// TIA Portal project "5 Run - 2 Stop (2T)" (V16)

(* hardware
DEVICE "S7-1200 station_1"  S7-1200 Station
   slot 0: "Rack_0"  S7-1200 Rack  Rack  V1.0
   slot 1: "PLC_1"  CPU 1212C AC/DC/Rly  6ES7 212-1BE40-0XB0  V4.0
*)

// ===== PLC "PLC_1"  CPU 1212C AC/DC/Rly =====

VAR_GLOBAL   // PLC tag table "Default tag table"
   "start1" AT %I0.2 : Bool;
   "K1" AT %Q0.0 : Bool;
   "stop1" AT %I0.4 : Bool;
   "k2" AT %Q0.1 : Bool;
   "start2" AT %I0.3 : Bool;
   "T1 tag" AT %M0.0 : Bool;
   "T2 tag" AT %M0.1 : Bool;
   "X" AT %M0.2 : Bool;
   "stop 2S" AT %M1.0 : Bool;
   "tag_2" AT %M1.1 : Bool;
   "K3" AT %Q0.2 : Bool;
   "T3 tag" AT %M0.3 : Bool;
END_VAR

// folder: System blocks/Program resources

DATA_BLOCK "T1"   // DB2
{ S7_Optimized_Access := 'TRUE' }
AUTHOR : Simatic
FAMILY : IEC
NAME : IEC_TMR
VERSION : 1.0
// stored: InstanceOfName IEC_TIMER
"IEC_TIMER"
BEGIN
END_DATA_BLOCK

DATA_BLOCK "T2"   // DB3
{ S7_Optimized_Access := 'TRUE' }
AUTHOR : Simatic
FAMILY : IEC
NAME : IEC_TMR
VERSION : 1.0
// stored: InstanceOfName IEC_TIMER
"IEC_TIMER"
BEGIN
END_DATA_BLOCK

// folder: (top level)

ORGANIZATION_BLOCK "Main"   // OB1, LAD, ProgramCycle
TITLE = "Main Program Sweep (Cycle)"
{ S7_Optimized_Access := 'TRUE' }
VERSION : 0.1
   VAR_INPUT
      Initial_Call : Bool;   // Initial call of this OB
      Remanence : Bool;   // =True, if remanent data are available
   END_VAR
BEGIN

REGION Network 1: start
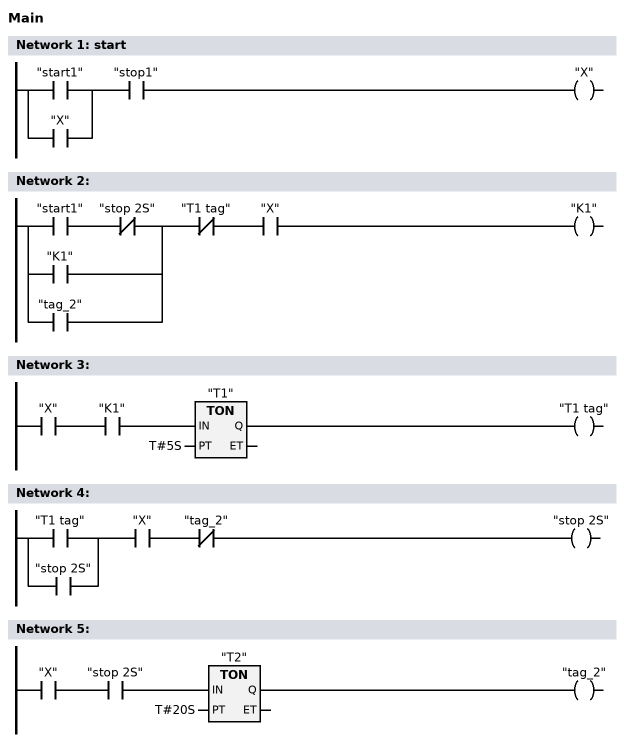
   RUNG wire#powerrail
      Contact( "start1" )
      wire#w1
      Contact( "stop1" )
      Coil( "X" )
   END_RUNG
   RUNG wire#powerrail
      Contact( "X" )
   END_RUNG wire#w1
   // the same network as SCL:
   "X" := ("start1" OR "X") AND "stop1";
END_REGION

REGION Network 2
   RUNG wire#powerrail
      Contact( "start1" )
      I_Contact( "stop 2S" )
      wire#w1
      I_Contact( "T1 tag" )
      Contact( "X" )
      Coil( "K1" )
   END_RUNG
   RUNG wire#powerrail
      Contact( "K1" )
   END_RUNG wire#w1
   RUNG wire#powerrail
      Contact( "tag_2" )
   END_RUNG wire#w1
   // the same network as SCL:
   "K1" := (("start1" AND NOT "stop 2S") OR "K1" OR "tag_2") AND NOT "T1 tag" AND "X";
END_REGION

REGION Network 3
   "T1".TON(IN := "X" AND "K1", PT := T#5S);
   "T1 tag" := "T1".Q;
END_REGION

REGION Network 4
   RUNG wire#powerrail
      Contact( "T1 tag" )
      wire#w1
      Contact( "X" )
      I_Contact( "tag_2" )
      Coil( "stop 2S" )
   END_RUNG
   RUNG wire#powerrail
      Contact( "stop 2S" )
   END_RUNG wire#w1
   // the same network as SCL:
   "stop 2S" := ("T1 tag" OR "stop 2S") AND "X" AND NOT "tag_2";
END_REGION

REGION Network 5
   "T2".TON(IN := "X" AND "stop 2S", PT := T#20S);
   "tag_2" := "T2".Q;
END_REGION
END_ORGANIZATION_BLOCK